SUBAPPLICATION Q_ChildPosition_AR_Bargraph_LeftToRight (* Bargraph Type 0 (LeftToRight): Skaliert AR-Eingang mit ScalePx und positioniert Child horizontal (X = Value x ScalePx, Y = 0) *)
  (* Standard: 61499-2; Description: Copyright (c) 2026 Meisterschulen am Ostbahnhof This program and the accompanying materials are made available under the terms of the Eclipse Public License 2.0 which is available at https://www.eclipse.org/legal/epl-2.0/ SPDX-License-Identifier: EPL-2.0 *)
  (* Version 1.0, 2026-09-27, Franz Höpfinger, Meisterschulen am Ostbahnhof, initial API and implementation: AR_R_MUL + Q_ChildPosition_AR_Horizontal *)
  PACKAGE MyLib::sys;
  IMPORT isobus::UT::Q::const::IDs::ID_NULL;
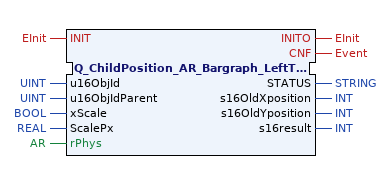
  EVENT_INPUT
    INIT : EInit; (* Service Initialization *)
  END_EVENT
  EVENT_OUTPUT
    INITO : EInit; (* Initialization Confirm *)
    CNF; (* Confirmation of Requested Service *)
  END_EVENT
  VAR_INPUT
    u16ObjId : UINT := ID_NULL; (* Object ID *)
    u16ObjIdParent : UINT := ID_NULL; (* Parent object ID *)
    xScale : BOOL := TRUE; (* FALSE = bypass. TRUE (default) = scale by DM/SKM factor for u16ObjIdParent. *)
    ScalePx : REAL := REAL#1.0; (* Pixel pro Werteinheit (Multiplikationsfaktor) *)
  END_VAR
  VAR_OUTPUT
    STATUS : STRING; (* Service Status - passthrough from the internal Q_ChildPosition *)
    s16OldXposition : INT; (* Old X position - passthrough from the internal Q_ChildPosition *)
    s16OldYposition : INT; (* Old Y position - passthrough from the internal Q_ChildPosition *)
    s16result : INT; (* retval - passthrough from the internal Q_ChildPosition, see Q_ChildPosition *)
  END_VAR
  SOCKETS
    rPhys : adapter::types::unidirectional::AR; (* Physical REAL value input (skaliert und auf X-Position abgebildet) *)
  END_SOCKETS
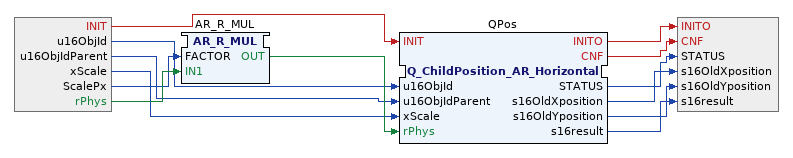
  SUBAPPS
    AR_R_MUL : MyLib::sys::AR_R_MUL;
    QPos : MyLib::sys::Q_ChildPosition_AR_Horizontal;
  END_SUBAPPS
  EVENT_CONNECTIONS
    INIT TO QPos.INIT;
    QPos.INITO TO INITO;
    QPos.CNF TO CNF;
  END_CONNECTIONS
  DATA_CONNECTIONS
    ScalePx TO AR_R_MUL.FACTOR;
    u16ObjId TO QPos.u16ObjId;
    u16ObjIdParent TO QPos.u16ObjIdParent;
    xScale TO QPos.xScale;
    QPos.STATUS TO STATUS;
    QPos.s16OldXposition TO s16OldXposition;
    QPos.s16OldYposition TO s16OldYposition;
    QPos.s16result TO s16result;
  END_CONNECTIONS
  ADAPTER_CONNECTIONS
    rPhys TO AR_R_MUL.IN1;
    AR_R_MUL.OUT TO QPos.rPhys;
  END_CONNECTIONS
END_SUBAPPLICATION
